// SIMATIC S7-200 SMART project (STEP 7-Micro/WIN SMART), CPU SR20

SYMBOL_TABLE Table 1
Symbol_38        M0.4
Symbol_37        M0.6
Symbol_36        V50.1
Symbol_35        V50.0
Symbol_34        T34
Symbol_33        T36
Symbol_32        T35
Symbol_31        M24.0
Symbol_30        M20.3
Symbol_29        T104
Symbol_28        M201.1
Symbol_27        T103
Symbol_26        T102
Symbol_25        M22.0
Symbol_24        M20.2
Symbol_23        T101
Symbol_22        M20.1
Symbol_21        T100
Symbol_20        M20.0
Symbol_19        T99
Symbol_18        T98
Symbol_17        T97
Symbol_16        T32
Symbol_15        MB16
Symbol_14        MB15
Symbol_13        VB30
Symbol_12        M11.0
Symbol_11        M10.6
Symbol_10        M10.4
Symbol_9         M10.3
Symbol_8         MB14
Symbol_7         VB50
Symbol_6         MB30
Symbol_5         M10.2
Symbol_4         VB20
Symbol_3         VW20
Symbol_2         MB12
Symbol_1         M10.1
Symbol_0         M10.0
END_SYMBOL_TABLE

SYMBOL_TABLE System Symbols
Always_On        SM0.0    // Always ON
END_SYMBOL_TABLE

ORGANIZATION_BLOCK MAIN:OB1
TITLE=Program Comments
BEGIN
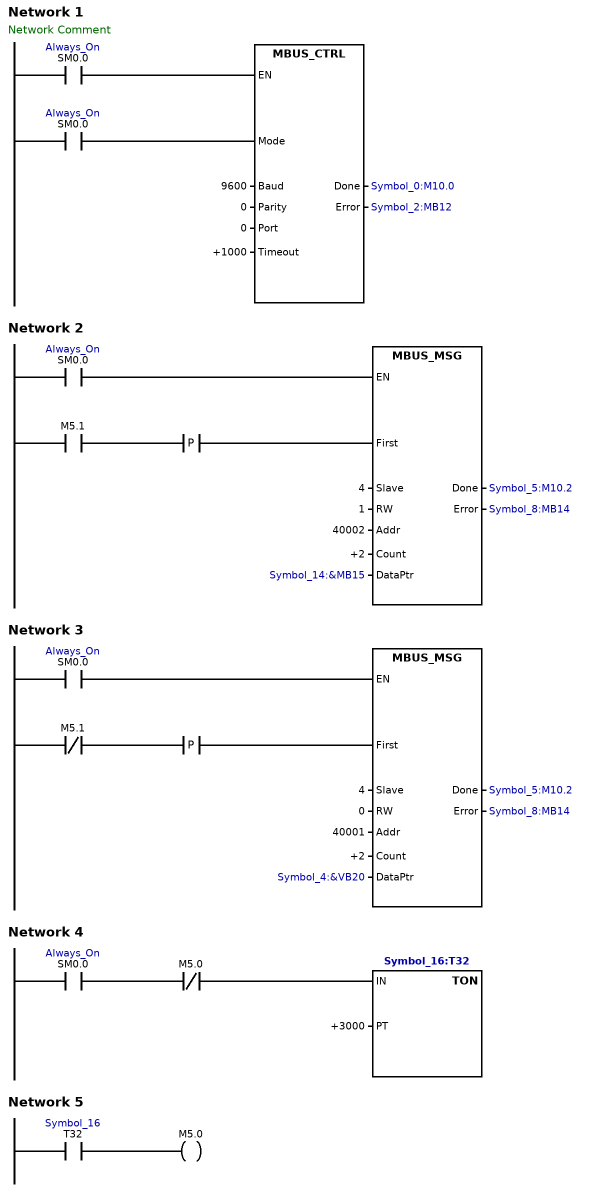
Network 1
// Network Comment
LD     Always_On:SM0.0
=      L60.0
LD     Always_On:SM0.0
=      L63.7
LD     L60.0
CALL   MBUS_CTRL:SBR1, L63.7, 9600, 0, 0, +1000, Symbol_0:M10.0, Symbol_2:MB12
Network 2
LD     Always_On:SM0.0
=      L60.0
LD     M5.1
EU
=      L63.7
LD     L60.0
CALL   MBUS_MSG:SBR2, L63.7, 4, 1, 40002, +2, &Symbol_14:MB15, Symbol_5:M10.2, Symbol_8:MB14
Network 3
LD     Always_On:SM0.0
=      L60.0
LDN    M5.1
EU
=      L63.7
LD     L60.0
CALL   MBUS_MSG:SBR2, L63.7, 4, 0, 40001, +2, &Symbol_4:VB20, Symbol_5:M10.2, Symbol_8:MB14
Network 4
LD     Always_On:SM0.0
AN     M5.0
TON    Symbol_16:T32, +3000
Network 5
LD     Symbol_16:T32
=      M5.0
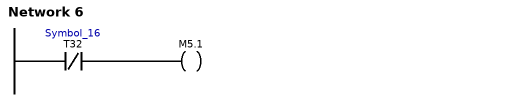
Network 6
LDN    Symbol_16:T32
=      M5.1
END_ORGANIZATION_BLOCK

// SBR1: protected block, not included

// SBR2: protected block, not included

// SBR3: protected block, not included
